VISUALIZATION Visualization  // 2x2
END_VISUALIZATION

(* stored: Version 1.1.0.1, ProductVersion 3.1.4024.6
   Visu Visualization: Id {90ac5b16-b2f9-4303-bd81-6d9e44072aea} *)
